TYPE LightConfigs :
STRUCT	
	ArduinoLightConfig : ArduinoLightConfig;
	EvosensLightConfig : EvosensLightConfig;
END_STRUCT
END_TYPE

(* stored: Version 1.1.0.1, ProductVersion 3.1.4024.12
   DUT LightConfigs: Id {bf6ec865-a6c5-49ab-a052-5e6fddbc13e9} *)
